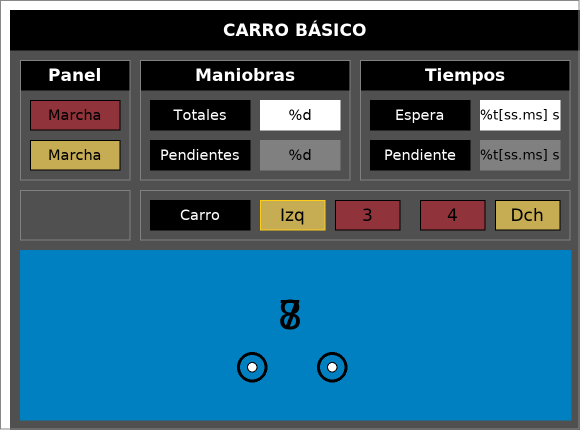
VISUALIZATION V_Carro  // 580x430
    Rectangle (10,50 570x380)
    Rectangle (140,190 430x50)
    Rectangle (20,60 110x30), "Panel"
    Rectangle (20,60 110x120)
    Rectangle (360,60 210x30), "Tiempos"
    Rectangle (360,60 210x120)
    Rectangle (10,10 570x40), "CARRO BÁSICO"
    RoundedRectangle (370,100 100x30), "Espera"
    Rectangle (140,60 210x30), "Maniobras"
    Rectangle (480,100 80x30), "%t[ss.ms] s", text variable: MAIN.Carro.TiempoEspera
        OnMouseClick: write the text variable via Default
    RoundedRectangle (370,140 100x30), "Pendiente"
    Rectangle (480,140 80x30), "%t[ss.ms] s", text variable: MAIN.Carro.TiempoPendiente
        OnMouseClick: write the text variable via Default
    Rectangle (30,100 90x30), "Marcha", colour toggle: MAIN.Carro.o_LamparaMarcha
        tap MAIN.Carro.o_LamparaMarcha
    Rectangle (30,140 90x30), "Marcha", colour toggle: MAIN.Carro.i_PulsadorMarcha
        toggle MAIN.Carro.i_PulsadorMarcha
    Rectangle (140,60 210x120)
    RoundedRectangle (150,100 100x30), "Totales"
    Rectangle (260,100 80x30), "%d", text variable: MAIN.Carro.ManiobrasTotales
        OnMouseClick: write the text variable via Default
    RoundedRectangle (150,140 100x30), "Pendientes"
    Rectangle (260,140 80x30), "%d", text variable: MAIN.Carro.ManiobrasPendientes
        OnMouseClick: write the text variable via Default
    Rectangle (20,250 551x170)
    Polyline (477,390)
    Polygon (105,385), colour toggle: MAIN.Carro.i_FinalCarreraIzquierda
        p2738717112: SEL (MAIN.Carro.i_FinalCarreraIzquierda, 0, 5)
        toggle MAIN.Carro.i_FinalCarreraIzquierda
    Polygon (435,385), colour toggle: MAIN.Carro.i_FinalCarreraDerecha
        p2738717112: SEL (MAIN.Carro.i_FinalCarreraDerecha, 0, 5)
        toggle MAIN.Carro.i_FinalCarreraDerecha
    Group (211,281 158x98), invisible if: MAIN.Carro.i_FinalCarreraIzquierda AND MAIN.Carro.i_FinalCarreraDerecha
        p3560616238: SEL (MAIN.Carro.i_FinalCarreraDerecha, SEL (MAIN.Carro.i_FinalCarreraIzquierda, 0, -125), 125)
        Polygon (0,0)
        Polygon (115,80)
        Group (106,71 28x28)
            Ellipse (0,0 30x30)
            Ellipse (10,10 10x10)
        Polygon (35,80)
        Group (26,71 28x28)
            Ellipse (0,0 30x30)
            Ellipse (10,10 10x10)
    Rectangle (270,295 40x40), "8", tooltip "Marcha derecha", invisible if: NOT MAIN.Carro.o_MarchaDerecha
        p3560616238: SEL (MAIN.Carro.i_FinalCarreraDerecha, SEL (MAIN.Carro.i_FinalCarreraIzquierda, 0, -125), 125)
    Rectangle (270,295 40x40), "7", invisible if: NOT MAIN.Carro.o_MarchaIzquierda
        p3560616238: SEL (MAIN.Carro.i_FinalCarreraDerecha, SEL (MAIN.Carro.i_FinalCarreraIzquierda, 0, -125), 125)
    RoundedRectangle (150,200 100x30), "Carro"
    Rectangle (335,200 65x30), "3", colour toggle: MAIN.Carro.o_MarchaIzquierda
        toggle MAIN.Carro.o_MarchaIzquierda
    Rectangle (420,200 65x30), "4", colour toggle: MAIN.Carro.o_MarchaDerecha
        toggle MAIN.Carro.o_MarchaDerecha
    Rectangle (260,200 65x30), "Izq", colour toggle: MAIN.Carro.i_FinalCarreraIzquierda
        toggle MAIN.Carro.i_FinalCarreraIzquierda
    Rectangle (495,200 65x30), "Dch", colour toggle: MAIN.Carro.i_FinalCarreraDerecha
        toggle MAIN.Carro.i_FinalCarreraDerecha
    Rectangle (20,190 110x50)
END_VISUALIZATION

(* stored: Version 1.1.0.1, ProductVersion 3.1.4024.16
   Visu V_Carro: Id {6c0d6d31-cc65-4443-98e2-0ca17fddc298} *)
